// TIA Portal V20 export
TYPE "UDT_MTP_AnaManInt"
TITLE = MTPDataObjectSUCLibrary/DataAssembly/AdvAnaOp
   STRUCT
      VMan : Real := 0.0;   // Manual Value (relevant, if SrcManAct is true)
      VMax { ExternalWritable := 'False'} : Real := 100.0;   // Value High Limit
      VMin { ExternalWritable := 'False'} : Real := 0.0;   // Value Low Limit
      OSLevel : Byte := 16#00;   // OSLevel variable
      SrcChannel { ExternalWritable := 'False'} : Bool;   // Selection of the active SourceMode interaction channel 0:The operator switches (*Op) shall be used 1:The automatic switches (*Aut) shall be used
      SrcManAut { ExternalWritable := 'False'} : Bool;   // Set SourceMode to Manual by automatic interaction (relevant, if SrcChannel is true) 1:SourceMode is set to Manual 0:no operation
      SrcIntAut { ExternalWritable := 'False'} : Bool;   // Set SourceMode to Internal by automatic interaction (relevant, if SrcChannel is true) 1:SourceMode is set to Internal 0:no operation
      SrcIntOp : Bool;   // Set SourceMode to Internal by operator interaction (relevant, if SrcChannel is false) 0-->1:request to set OperationMode to Internal 1-->0:acknowledge by PEA
      SrcManOp : Bool;   // Set SourceMode to Manual by operator interaction (relevant, if SrcChannel is false) 0-->1:request to set OperationMode to Manual 1-->0:acknowledge by PEA
      SrcIntAct { ExternalWritable := 'False'} : Bool;   // 1: current mode is Internal 0: current mode is not Internal
      SrcManAct { ExternalWritable := 'False'} : Bool;   // 1: current mode is Manual 0: current mode is not Manual
      WQC { ExternalWritable := 'False'} : Byte := 16#FF;   // Worst Quality Code variable
      VOut { ExternalWritable := 'False'} : Real := 0.0;   // Value Output
      VSclMax { ExternalWritable := 'False'} : Real := 100.0;   // Value Scale High Limit
      VSclMin { ExternalWritable := 'False'} : Real := 0.0;   // Value Scale Low Limit
      VUnit { ExternalWritable := 'False'} : Int := 1001;   // Value Unit
      VInt { ExternalWritable := 'False'} : Real := 0.0;   // Internal Value(relevant, if SrcIntAct is true)
      VRbk { ExternalWritable := 'False'} : Real := 0.0;   // Readback Value
      VFbk { ExternalWritable := 'False'} : Real;   // Feedback Value
   END_STRUCT;
END_TYPE
